Fanuc KAREL source: SET_TSK_NAME.kl

PROGRAM T
%NOLOCKGROUP
VAR
 v0 : STRING[40]
 v1 : STRING[40]
 v2 : INTEGER
BEGIN
 SET_TSK_NAME(v0, v1, v2)
END T
